{attribute 'GeneratedUsingTerminal: EPP3632-0001-0016'}
{attribute addProperty BoxType "EPP3632-0001-0016"}
{attribute addProperty Id "StartTimeNextLatchAT %I*ULINT8"}
{attribute addProperty CRC "2600321653"}
{attribute addProperty Size "8"}
TYPE NextSync1Time_9AFDC275 :
STRUCT
	{attribute addProperty Name "StartTimeNextLatch"}
	StartTimeNextLatch AT %I* : ULINT;
END_STRUCT
END_TYPE

(* stored: Version 1.2.0.0, ProductVersion 3.1.4024.9
   DUT NextSync1Time_9AFDC275: Id {b1b89b7f-2708-470b-964b-a4258994acfe} *)
